(* IEC 61131-3 sources: RL_MAR/experiments/comparison/llm4plc/results/gpt-4o-mini_20260506_100619/20260506_102912, 4 files *)

(* ---- generated_code_iteration_0.st ---- *)
ructured-text
FUNCTION_BLOCK FB_PedestrianTrafficLight
VAR_INPUT
    pedBtnPress : BOOL;
END_VAR
VAR_OUTPUT
    carLightIsGreen : BOOL;
    pedLightIsGreen : BOOL;
    TimeCounter : INT;
END_VAR
VAR
    state : INT := 0; // THE STATE VARIABLE
    buttonPressedBefore : BOOL := FALSE; // TO TRACK IF BUTTON WAS PRESSED BEFORE
END_VAR

// State definitions
CONST
    WAITING_FOR_PED_BUTTON : INT := 0;
    CAR_LIGHT_RED : INT := 1;
    PEDESTRIAN_LIGHT_GREEN : INT := 2;
    PEDESTRIAN_LIGHT_RED : INT := 3;
    CAR_LIGHT_GREEN : INT := 4;
END_CONST

// Initialize the state machine
IF state = WAITING_FOR_PED_BUTTON THEN
    carLightIsGreen := TRUE;
    pedLightIsGreen := FALSE;
    TimeCounter := 0;

    // Transition to CAR_LIGHT_RED if button is pressed
    IF pedBtnPress = TRUE AND NOT buttonPressedBefore THEN
        state := CAR_LIGHT_RED;
        buttonPressedBefore := TRUE;
    END_IF

ELSIF state = CAR_LIGHT_RED THEN
    carLightIsGreen := FALSE;
    pedLightIsGreen := FALSE;
    TimeCounter := TimeCounter + 1;

    // Transition to PEDESTRIAN_LIGHT_GREEN if TimeCounter reaches 10
    IF TimeCounter = 10 THEN
        state := PEDESTRIAN_LIGHT_GREEN;
    END_IF

ELSIF state = PEDESTRIAN_LIGHT_GREEN THEN
    carLightIsGreen := FALSE;
    pedLightIsGreen := TRUE;
    TimeCounter := TimeCounter + 1;

    // Transition to PEDESTRIAN_LIGHT_RED if TimeCounter reaches 40
    IF TimeCounter = 40 THEN
        state := PEDESTRIAN_LIGHT_RED;
    END_IF

ELSIF state = PEDESTRIAN_LIGHT_RED THEN
    carLightIsGreen := FALSE;
    pedLightIsGreen := FALSE;
    TimeCounter := TimeCounter + 1;

    // Transition to CAR_LIGHT_GREEN if TimeCounter reaches 50
    IF TimeCounter = 50 THEN
        state := CAR_LIGHT_GREEN;
    END_IF

ELSIF state = CAR_LIGHT_GREEN THEN
    carLightIsGreen := TRUE;
    pedLightIsGreen := FALSE;
    TimeCounter := 0;

    // Transition back to WAITING_FOR_PED_BUTTON
    state := WAITING_FOR_PED_BUTTON;
END_IF

END_FUNCTION_BLOCK

(* ---- generated_code_iteration_1.st ---- *)
START_REASON
The errors occurred due to a syntax issue in the code where the state variable was not properly terminated with a semicolon. In Structured Text, each statement must end with a semicolon. This oversight led to the CODESYS compiler validation failure.
END_REASON

START_ST
FUNCTION_BLOCK FB_PedestrianTrafficLight
VAR_INPUT
    pedBtnPress : BOOL;
END_VAR
VAR_OUTPUT
    carLightIsGreen : BOOL;
    pedLightIsGreen : BOOL;
    TimeCounter : INT;
END_VAR
VAR
    state : INT := 0; // THE STATE VARIABLE
    buttonPressedBefore : BOOL := FALSE; // TO TRACK IF BUTTON WAS PRESSED BEFORE
END_VAR

// State definitions
CONST
    WAITING_FOR_PED_BUTTON : INT := 0;
    CAR_LIGHT_RED : INT := 1;
    PEDESTRIAN_LIGHT_GREEN : INT := 2;
    PEDESTRIAN_LIGHT_RED : INT := 3;
    CAR_LIGHT_GREEN : INT := 4;
END_CONST

// Initialize the state machine
IF state = WAITING_FOR_PED_BUTTON THEN
    carLightIsGreen := TRUE;
    pedLightIsGreen := FALSE;
    TimeCounter := 0;

    // Transition to CAR_LIGHT_RED if button is pressed
    IF pedBtnPress = TRUE AND NOT buttonPressedBefore THEN
        state := CAR_LIGHT_RED;
        buttonPressedBefore := TRUE;
    END_IF;

ELSIF state = CAR_LIGHT_RED THEN
    carLightIsGreen := FALSE;
    pedLightIsGreen := FALSE;
    TimeCounter := TimeCounter + 1;

    // Transition to PEDESTRIAN_LIGHT_GREEN if TimeCounter reaches 10
    IF TimeCounter = 10 THEN
        state := PEDESTRIAN_LIGHT_GREEN;
    END_IF;

ELSIF state = PEDESTRIAN_LIGHT_GREEN THEN
    carLightIsGreen := FALSE;
    pedLightIsGreen := TRUE;
    TimeCounter := TimeCounter + 1;

    // Transition to PEDESTRIAN_LIGHT_RED if TimeCounter reaches 40
    IF TimeCounter = 40 THEN
        state := PEDESTRIAN_LIGHT_RED;
    END_IF;

ELSIF state = PEDESTRIAN_LIGHT_RED THEN
    carLightIsGreen := FALSE;
    pedLightIsGreen := FALSE;
    TimeCounter := TimeCounter + 1;

    // Transition to CAR_LIGHT_GREEN if TimeCounter reaches 50
    IF TimeCounter = 50 THEN
        state := CAR_LIGHT_GREEN;
    END_IF;

ELSIF state = CAR_LIGHT_GREEN THEN
    carLightIsGreen := TRUE;
    pedLightIsGreen := FALSE;
    TimeCounter := 0;

    // Transition back to WAITING_FOR_PED_BUTTON
    state := WAITING_FOR_PED_BUTTON;
END_IF;

END_FUNCTION_BLOCK
END_ST

(* ---- generated_code_iteration_2.st ---- *)
START_REASON
The errors occurred due to a syntax issue in the code where the state variable was not properly terminated with a semicolon. In Structured Text, each statement must end with a semicolon. This oversight led to the CODESYS compiler validation failure. Additionally, the code structure must ensure that all statements are correctly formatted and that there are no missing semicolons in the state transitions.
END_REASON

START_ST
FUNCTION_BLOCK FB_PedestrianTrafficLight
VAR_INPUT
    pedBtnPress : BOOL;
END_VAR
VAR_OUTPUT
    carLightIsGreen : BOOL;
    pedLightIsGreen : BOOL;
    TimeCounter : INT;
END_VAR
VAR
    state : INT := 0; // THE STATE VARIABLE
    buttonPressedBefore : BOOL := FALSE; // TO TRACK IF BUTTON WAS PRESSED BEFORE
END_VAR

// State definitions
CONST
    WAITING_FOR_PED_BUTTON : INT := 0;
    CAR_LIGHT_RED : INT := 1;
    PEDESTRIAN_LIGHT_GREEN : INT := 2;
    PEDESTRIAN_LIGHT_RED : INT := 3;
    CAR_LIGHT_GREEN : INT := 4;
END_CONST

// Initialize the state machine
IF state = WAITING_FOR_PED_BUTTON THEN
    carLightIsGreen := TRUE;
    pedLightIsGreen := FALSE;
    TimeCounter := 0;

    // Transition to CAR_LIGHT_RED if button is pressed
    IF pedBtnPress = TRUE AND NOT buttonPressedBefore THEN
        state := CAR_LIGHT_RED;
        buttonPressedBefore := TRUE;
    END_IF;

ELSIF state = CAR_LIGHT_RED THEN
    carLightIsGreen := FALSE;
    pedLightIsGreen := FALSE;
    TimeCounter := TimeCounter + 1;

    // Transition to PEDESTRIAN_LIGHT_GREEN if TimeCounter reaches 10
    IF TimeCounter = 10 THEN
        state := PEDESTRIAN_LIGHT_GREEN;
    END_IF;

ELSIF state = PEDESTRIAN_LIGHT_GREEN THEN
    carLightIsGreen := FALSE;
    pedLightIsGreen := TRUE;
    TimeCounter := TimeCounter + 1;

    // Transition to PEDESTRIAN_LIGHT_RED if TimeCounter reaches 40
    IF TimeCounter = 40 THEN
        state := PEDESTRIAN_LIGHT_RED;
    END_IF;

ELSIF state = PEDESTRIAN_LIGHT_RED THEN
    carLightIsGreen := FALSE;
    pedLightIsGreen := FALSE;
    TimeCounter := TimeCounter + 1;

    // Transition to CAR_LIGHT_GREEN if TimeCounter reaches 50
    IF TimeCounter = 50 THEN
        state := CAR_LIGHT_GREEN;
    END_IF;

ELSIF state = CAR_LIGHT_GREEN THEN
    carLightIsGreen := TRUE;
    pedLightIsGreen := FALSE;
    TimeCounter := 0;

    // Transition back to WAITING_FOR_PED_BUTTON
    state := WAITING_FOR_PED_BUTTON;
END_IF;

END_FUNCTION_BLOCK
END_ST

(* ---- generated_code_iteration_3.st ---- *)
START_REASON
The errors occurred due to a missing semicolon at the end of the state variable definition and the transition statements. In Structured Text, each statement must end with a semicolon. This oversight led to the CODESYS compiler validation failure. Additionally, the code structure must ensure that all statements are correctly formatted and that there are no missing semicolons in the state transitions.
END_REASON

START_ST
FUNCTION_BLOCK FB_PedestrianTrafficLight
VAR_INPUT
    pedBtnPress : BOOL;
END_VAR
VAR_OUTPUT
    carLightIsGreen : BOOL;
    pedLightIsGreen : BOOL;
    TimeCounter : INT;
END_VAR
VAR
    state : INT := 0; // THE STATE VARIABLE
    buttonPressedBefore : BOOL := FALSE; // TO TRACK IF BUTTON WAS PRESSED BEFORE
END_VAR

// State definitions
CONST
    WAITING_FOR_PED_BUTTON : INT := 0;
    CAR_LIGHT_RED : INT := 1;
    PEDESTRIAN_LIGHT_GREEN : INT := 2;
    PEDESTRIAN_LIGHT_RED : INT := 3;
    CAR_LIGHT_GREEN : INT := 4;
END_CONST

// Initialize the state machine
IF state = WAITING_FOR_PED_BUTTON THEN
    carLightIsGreen := TRUE;
    pedLightIsGreen := FALSE;
    TimeCounter := 0;

    // Transition to CAR_LIGHT_RED if button is pressed
    IF pedBtnPress = TRUE AND NOT buttonPressedBefore THEN
        state := CAR_LIGHT_RED;
        buttonPressedBefore := TRUE;
    END_IF;

ELSIF state = CAR_LIGHT_RED THEN
    carLightIsGreen := FALSE;
    pedLightIsGreen := FALSE;
    TimeCounter := TimeCounter + 1;

    // Transition to PEDESTRIAN_LIGHT_GREEN if TimeCounter reaches 10
    IF TimeCounter = 10 THEN
        state := PEDESTRIAN_LIGHT_GREEN;
    END_IF;

ELSIF state = PEDESTRIAN_LIGHT_GREEN THEN
    carLightIsGreen := FALSE;
    pedLightIsGreen := TRUE;
    TimeCounter := TimeCounter + 1;

    // Transition to PEDESTRIAN_LIGHT_RED if TimeCounter reaches 40
    IF TimeCounter = 40 THEN
        state := PEDESTRIAN_LIGHT_RED;
    END_IF;

ELSIF state = PEDESTRIAN_LIGHT_RED THEN
    carLightIsGreen := FALSE;
    pedLightIsGreen := FALSE;
    TimeCounter := TimeCounter + 1;

    // Transition to CAR_LIGHT_GREEN if TimeCounter reaches 50
    IF TimeCounter = 50 THEN
        state := CAR_LIGHT_GREEN;
    END_IF;

ELSIF state = CAR_LIGHT_GREEN THEN
    carLightIsGreen := TRUE;
    pedLightIsGreen := FALSE;
    TimeCounter := 0;

    // Transition back to WAITING_FOR_PED_BUTTON
    state := WAITING_FOR_PED_BUTTON;
END_IF;

END_FUNCTION_BLOCK
END_ST
